	                #sFB_RightAngledTransfer421(iUDT_Configuration := #iUDT_Configuration."421".RightAngledTransfer,
	                                            iUDT_LowerConveyorConfiguration := #iUDT_Configuration."420".Conveyor,
	                                            iUDT_UpperConveyorConfiguration := #iUDT_Configuration."421".Conveyor,
	                                            iUDT_PECConfiguration := #iUDT_Configuration."420".PEC_EoS,
	                                            ii_DestinationA := 0,
	                                            ii_DestinationB := 0,
	                                            ii_DestinationC := 0,
	                                            ii_DestinationD := 1,
	                                            ix_HardwareOk := #iUDT_HardwareOk."420",
	                                            ix_400vOk := #ix_400vOk,
	                                            ix_24vOk := #ix_24vOk,
	                                            ix_SafetyOk := #ix_SafetyOk,
	                                            ix_AirPressureOk := #ix_AirPressureOk,
	                                            ix_SectionIsDown := #sFB_MCOConveyLinxAixController420.sUDT_AixInputsFullModule.AllSensorPortInputs.RightPin2,
	                                            ix_SectionIsUp := #sFB_MCOConveyLinxAixController420.sUDT_AixInputsFullModule.AllSensorPortInputs.RightSensor,
	                                            ix_ConveyorAAuto := FALSE,
	                                            ix_ConveyorBAuto := #iqUDT_WorkstationCommonStatus."430".AutoON,
	                                            ix_ConveyorCAuto := FALSE,
	                                            ix_ConveyorDAuto := #iqUDT_WorkstationCommonStatus."410".AutoON,
	                                            ix_PEC := #sFB_MCOConveyLinxAixController420.sUDT_AixInputsFullModule.AllSensorPortInputs.LeftSensor,
	                                            ix_ExternalReceiveRequestA := FALSE,
	                                            ix_ExternalReceiveRequestB := FALSE,
	                                            ix_ExternalReceiveRequestC := FALSE,
	                                            ix_ExternalReceiveRequestD := NOT #iqUDT_WorkstationStatus."410".PEC_EoS.PEC,
	                                            ix_PECInfeedA := false,
	                                            ix_PECInfeedD := #iqUDT_WorkstationStatus."410".PEC_EoS.PEC,
	                                            qUDT_HMIRATStatus => #iqUDT_WorkstationStatus."421".RightAngledTransfer,
	                                            qUDT_HMIConveyorStatus => #iqUDT_WorkstationStatus."420".Conveyor,
	                                            qUDT_HMIPECStatus => #iqUDT_WorkstationStatus."421".PEC_EoS,
	                                            qUDT_RATStatus => #iqUDT_WorkstationCommonStatus."421",
	                                            qUDT_ConveyorStatus => #iqUDT_WorkstationCommonStatus."420",
	                                            qx_PopupControl => #qx_PopupControl421,
	                                            qx_ExternalSendRequestA => #tx_dummy,
	                                            qx_ExternalSendRequestB => #tx_dummy,
	                                            qx_ExternalSendRequestC => #tx_dummy,
	                                            qx_ExternalSendRequestD => #tx_dummy,
	                                            iqUDT_EquipmentControl := #iqUDT_EquipmentControlFirstStation,
	                                            iqUDT_RATCommand := #iqUDT_WorkstationCommands."421".RightAngledTransfer,
	                                            iqUDT_ConveyorCommand := #iqUDT_WorkstationCommands."420".Conveyor,
	                                            iqUDT_RATStatistics := #iqUDT_WorkstationStatistics."421".RightAngledTransfer,
	                                            iqUDT_ConveyorStatistics := #iqUDT_WorkstationStatistics."420".Conveyor,
	                                            iqUDT_PECStatistics := #iqUDT_WorkstationStatistics."421".PEC_EoS,
	                                            iqUDT_HandShakeConveyorA := #tUDT_dummyHandshake,
	                                            iqUDT_HandShakeConveyorB := #sUDT_Handshake420,
	                                            iqUDT_HandShakeConveyorC := #tUDT_dummyHandshake,
	                                            iqUDT_HandShakeConveyorD := #sUDT_Handshake410,
	                                            iqUDT_LowerConveyorInterface := #sUDT_Interface420,
	                                            iqUDT_UpperConveyorInterface := #sUDT_Interface421,
	                                            iqUDT_RATPositioning := #iqUDT_RATPositioning420,
	                                            iqUDT_BladeStopEoSInterface := #tudt_Bladeinterfacedummy,
	                                            iqUDT_BladeStopBoSInterface := #tudt_Bladeinterfacedummy);

	            END_REGION

	            REGION MCO

	                #sFB_MCOConveyLinxAixController421(iUDT_AixConfig := #iUDT_Configuration."421".MCO_M01,
	                                                   iv_AixInputsModule := #iv_MotorInput420,
	                                                   ii_PositionSetpoint := #iqUDT_RATPositioning420.Upper.EndPosition,
	                                                   ix_24vOk := #ix_24vOk,
	                                                   ix_SimulationModeActive := "DB_Memory".Simulation,
	                                                   ii_MotorPositionId := 2,
	                                                   ix_StartPositioning := #iqUDT_RATPositioning420.Upper.Start,
	                                                   ix_ResetPosition := #iqUDT_RATPositioning420.Upper.ResetPosition,
	                                                   qUDT_HMIStatus => #iqUDT_WorkstationStatus."421".MCO_M01,
	                                                   qx_Positioned => #iqUDT_RATPositioning420.Upper.Done,
	                                                   iqv_AixOutputsModule := #iqv_MotorOutput420,
	                                                   iqUDT_ConveyorInterface := #sUDT_Interface421,
	                                                   iqUDT_MCOStatistics := #iqUDT_WorkstationStatistics."421".MCO_M01);
	            END_REGION

	        END_REGION

	        REGION 430
	            REGION ZPA First conveyor

	                #sFB_ZpaFirstConveyor430(iUDT_AixInputsModule := #iUDT_InputsModule430,
	                                         iUDT_AixZpaConfig := #iUDT_Configuration."430".Conveyor,
	                                       ix_24vOk := NOT #ix_24vOk,
	                                       ix_HardwareOk := #iUDT_HardwareOk."430",
	                                       ix_SimulationModeActive := "DB_Memory".Simulation,
	                                       qUDT_AixOutputsModule => #qUDT_OutputsModule430,
	                                       iqUDT_ZPAinterface := #sUDT_ZPAinterface430,
	                                       iqUDT_PecStatus := #iqUDT_WorkstationStatus."430".PEC_EoS,
	                                       iqUDT_ZpaControllerStatus := #iqUDT_WorkstationStatus."430".MCO_ZPA,
	                                       iqUDT_HandShakeUp := #sUDT_Handshake430);
	            END_REGION

	            REGION ZPA Zone status

	                #sFB_ZpaStatus430(ii_ModuleID := 1,
	                                        iqUDT_PecStatus := #iqUDT_WorkstationStatus."430".PEC_EoS,
	                                        iqUDT_ZpaControllerStatus := #iqUDT_WorkstationStatus."430".MCO_ZPA,
	                                        iqUDT_ZPAInterface := #sUDT_ZPAinterface430,
	                                        qUDT_ConveyorStatus => #iqUDT_WorkstationStatus."430".Conveyor);

	            END_REGION
	        END_REGION

	        REGION 440
	            REGION ZPA Zone status

	                #sFB_ZpaStatus440(ii_ModuleID := 1,
	                                        iqUDT_PecStatus := #iqUDT_WorkstationStatus."440".PEC_EoS,
	                                        iqUDT_ZpaControllerStatus := #iqUDT_WorkstationStatus."440".MCO_ZPA,
	                                        iqUDT_ZPAInterface := #sUDT_ZPAinterface430,
	                                        qUDT_ConveyorStatus => #iqUDT_WorkstationStatus."440".Conveyor);

	            END_REGION
	        END_REGION

	        REGION 450
	            REGION ZPA Zone status

	                #sFB_ZpaStatus450(ii_ModuleID := 2,
	                                        iqUDT_PecStatus := #iqUDT_WorkstationStatus."450".PEC_EoS,
	                                        iqUDT_ZpaControllerStatus := #iqUDT_WorkstationStatus."450".MCO_ZPA,
	                                        iqUDT_ZPAInterface := #sUDT_ZPAinterface430,
	                                        qUDT_ConveyorStatus => #iqUDT_WorkstationStatus."450".Conveyor);

	            END_REGION
	        END_REGION

	        REGION 260
	            REGION ZPA Zone status

	                #sFB_ZpaStatus460(ii_ModuleID := 2,
	                                        iqUDT_PecStatus := #iqUDT_WorkstationStatus."260".PEC_EoS,
	                                        iqUDT_ZpaControllerStatus := #iqUDT_WorkstationStatus."260".MCO_ZPA,
	                                        iqUDT_ZPAInterface := #sUDT_ZPAinterface230,
	                                        qUDT_ConveyorStatus => #iqUDT_WorkstationStatus."260".Conveyor);

	            END_REGION
	        END_REGION

	        REGION 470
	            REGION ZPA Zone status

	                #sFB_ZpaStatus470(ii_ModuleID := 3,
	                                        iqUDT_PecStatus := #iqUDT_WorkstationStatus."470".PEC_EoS,
	                                        iqUDT_ZpaControllerStatus := #iqUDT_WorkstationStatus."470".MCO_ZPA,
	                                        iqUDT_ZPAInterface := #sUDT_ZPAinterface430,
	                                        qUDT_ConveyorStatus => #iqUDT_WorkstationStatus."470".Conveyor);

	            END_REGION
	        END_REGION

	        REGION 480
	            REGION ZPA Last conveyor

	                #sFB_ZpaLastConveyor480(iUDT_AixInputsModule := #iUDT_InputsModule470,
	                                        iUDT_AixZpaConfig := #iUDT_Configuration."480".Conveyor,
	                                      ix_SafetyOk := #ix_SafetyOk,
	                                      ix_24vOk := #ix_24vOk,
	                                      ix_HardwareOk := #iUDT_HardwareOk."480",
	                                      ix_SimulationModeActive := "DB_Memory".Simulation,
	                                      qUDT_AixOutputsModule => #qUDT_OutputsModule470,
	                                      qUDT_CommonStatus => #iqUDT_WorkstationCommonStatus."480",
	                                      iqUDT_EquipmentControl := #iqUDT_EquipmentControlSecondStation,
	                                      iqUDT_ZPACommand := #iqUDT_WorkstationCommands."480".SegmentZPA,
	                                      iqUDT_ZPAinterface := #sUDT_ZPAinterface430,
	                                      iqUDT_PecStatus := #iqUDT_WorkstationStatus."480".PEC_EoS,
	                                      iqUDT_ZpaControllerStatus := #iqUDT_WorkstationStatus."480".MCO_ZPA,
	                                      iqUDT_Handshake := #sUDT_Handshake480);
	            END_REGION

	            REGION ZPA Zone status

	                #sFB_ZpaStatus480(ii_ModuleID := 3,
	                                        iqUDT_PecStatus := #iqUDT_WorkstationStatus."280".PEC_EoS,
	                                        iqUDT_ZpaControllerStatus := #iqUDT_WorkstationStatus."280".MCO_ZPA,
	                                        iqUDT_ZPAInterface := #sUDT_ZPAinterface230,
	                                        qUDT_ConveyorStatus => #iqUDT_WorkstationStatus."280".Conveyor);

	            END_REGION

	            REGION Barcode Scanner
	                #sFB_Scanner_481(iUDT_ScannerInput := #iUDT_ScannerInput501,
	                                 iUDT_ScannerConfiguration := #iUDT_Configuration."481",
	                                 iUDT_ConveyorInterface := #sUDT_Interface480,
	                                 ix_24vOk := TRUE,
	                                 ix_HardwareOk := TRUE,
	                                 ix_SimulationModeActive := FALSE,
	                                 ix_CloseWindow := #iqUDT_WorkstationStatus."480".PEC_EoS.PEC,
	                                 ix_Trigger := NOT #iqUDT_WorkstationStatus."480".PEC_EoS.PEC,
	                                 qUDT_ScannerOutput => #qUDT_ScannerOutput501,
	                                 qUDT_HMIStatus => #iqUDT_WorkstationStatus."481",
	                                 qUDT_CommonStatus => #iqUDT_WorkstationCommonStatus."481",
	                                 qs_Barcode => #ts_Barcode481,
	                                 iqUDT_Statistics := #iqUDT_WorkstationStatistics."481",
	                                 iqUDT_EquipmentControl := #iqUDT_EquipmentControlSecondStation);
	            END_REGION
	        END_REGION

	        REGION 490

	            REGION Displacement
	                #sFB_Displacement490(#sUDT_Interface490);
	            END_REGION

	            REGION MCO

	                #sFB_MCOConveyLinxAixController490(iUDT_AixConfig := #iUDT_Configuration."490".MCO_M01,
	                                                   iv_AixInputsModule := #iv_MotorInput490,
	                                                   ii_PositionSetpoint := #iqUDT_RATPositioning490.Lower.EndPosition,
	                                                   ix_24vOk := #ix_24vOk,
	                                                   ix_SimulationModeActive := "DB_Memory".Simulation,
	                                                   ii_MotorPositionId := 1,
	                                                   ix_StartPositioning := #iqUDT_RATPositioning490.Lower.Start,
	                                                   ix_ResetPosition := #iqUDT_RATPositioning490.Lower.ResetPosition,
	                                                   qUDT_HMIStatus => #iqUDT_WorkstationStatus."490".MCO_M01,
	                                                   qx_Positioned => #iqUDT_RATPositioning490.Lower.Done,
	                                                   iqv_AixOutputsModule := #iqv_MotorOutput490,
	                                                   iqUDT_ConveyorInterface := #sUDT_Interface490,
	                                                   iqUDT_MCOStatistics := #iqUDT_WorkstationStatistics."490".MCO_M01);
	            END_REGION
	        END_REGION


	        REGION 491

	            REGION Displacement
	                #sFB_Displacement491(#sUDT_Interface491);
	            END_REGION

	            REGION RAT

	                #sFB_RightAngledTransfer491(iUDT_Configuration := #iUDT_Configuration."491".RightAngledTransfer,
	                                            iUDT_LowerConveyorConfiguration := #iUDT_Configuration."490".Conveyor,
	                                            iUDT_UpperConveyorConfiguration := #iUDT_Configuration."491".Conveyor,
	                                            iUDT_PECConfiguration := #iUDT_Configuration."490".PEC_EoS,
	                                            ii_DestinationA := #si_DestinationA491,
	                                            ii_DestinationB := 0,
	                                            ii_DestinationC := 0,
	                                            ii_DestinationD := 0,
	                                            ix_HardwareOk := #iUDT_HardwareOk."490",
	                                            ix_400vOk := #ix_400vOk,
	                                            ix_24vOk := #ix_24vOk,
	                                            ix_SafetyOk := #ix_SafetyOk,
	                                            ix_AirPressureOk := #ix_AirPressureOk,
	                                            ix_SectionIsDown := #sFB_MCOConveyLinxAixController490.sUDT_AixInputsFullModule.AllSensorPortInputs.RightPin2,
	                                            ix_SectionIsUp := #sFB_MCOConveyLinxAixController490.sUDT_AixInputsFullModule.AllSensorPortInputs.RightSensor,
	                                            ix_ConveyorAAuto := #iqUDT_WorkstationCommonStatus."480".AutoON,
	                                            ix_ConveyorBAuto := FALSE,
	                                            ix_ConveyorCAuto := FALSE,
	                                            ix_ConveyorDAuto := #iqUDT_WorkstationCommonStatus."500".AutoON,
	                                            ix_PEC := #sFB_MCOConveyLinxAixController490.sUDT_AixInputsFullModule.AllSensorPortInputs.LeftSensor,
	                                            ix_ExternalReceiveRequestA := NOT #iqUDT_WorkstationStatus."480".PEC_EoS.PEC,
	                                            ix_ExternalReceiveRequestB := FALSE,
	                                            ix_ExternalReceiveRequestC := FALSE,
	                                            ix_ExternalReceiveRequestD := FALSE,
	                                            ix_PECInfeedA := #iqUDT_WorkstationStatus."480".PEC_EoS.PEC,
	                                            qUDT_HMIRATStatus => #iqUDT_WorkstationStatus."491".RightAngledTransfer,
	                                            qUDT_HMIConveyorStatus => #iqUDT_WorkstationStatus."490".Conveyor,
	                                            qUDT_HMIPECStatus => #iqUDT_WorkstationStatus."491".PEC_EoS,
	                                            qUDT_RATStatus => #iqUDT_WorkstationCommonStatus."491",
	                                            qUDT_ConveyorStatus => #iqUDT_WorkstationCommonStatus."490",
	                                            qx_PopupControl => #qx_PopupControl491,
	                                            qx_ExternalSendRequestA => #tx_dummy,
	                                            qx_ExternalSendRequestB => #tx_dummy,
	                                            qx_ExternalSendRequestC => #tx_dummy,
	                                            qx_ExternalSendRequestD => #tx_dummy,
	                                            iqUDT_EquipmentControl := #iqUDT_EquipmentControlFirstStation,
	                                            iqUDT_RATCommand := #iqUDT_WorkstationCommands."491".RAT,
	                                            iqUDT_ConveyorCommand := #iqUDT_WorkstationCommands."490".Conveyor,
	                                            iqUDT_RATStatistics := #iqUDT_WorkstationStatistics."491".RightAngledTransfer,
	                                            iqUDT_ConveyorStatistics := #iqUDT_WorkstationStatistics."490".Conveyor,
	                                            iqUDT_PECStatistics := #iqUDT_WorkstationStatistics."491".PEC_EoS,
	                                            iqUDT_HandShakeConveyorA := #sUDT_Handshake480,
	                                            iqUDT_HandShakeConveyorB := #tUDT_dummyHandshake,
	                                            iqUDT_HandShakeConveyorC := #tUDT_dummyHandshake,
	                                            iqUDT_HandShakeConveyorD := #sUDT_Handshake491,
	                                            iqUDT_LowerConveyorInterface := #sUDT_Interface490,
	                                            iqUDT_UpperConveyorInterface := #sUDT_Interface491,
	                                            iqUDT_RATPositioning := #iqUDT_RATPositioning490,
	                                            iqUDT_BladeStopEoSInterface := #tudt_Bladeinterfacedummy,
	                                            iqUDT_BladeStopBoSInterface := #tudt_Bladeinterfacedummy);



	            END_REGION

	            REGION MCO

	                #sFB_MCOConveyLinxAixController491(iUDT_AixConfig := #iUDT_Configuration."491".MCO_M01,
	                                                   iv_AixInputsModule := #iv_MotorInput490,
	                                                   ix_24vOk := #ix_24vOk,
	                                                   ix_SimulationModeActive := "DB_Memory".Simulation,
	                                                   ii_MotorPositionId := 2,
	                                                   qUDT_HMIStatus => #iqUDT_WorkstationStatus."491".MCO_M01,
	                                                   iqv_AixOutputsModule := #iqv_MotorOutput490,
	                                                   iqUDT_ConveyorInterface := #sUDT_Interface491,
	                                                   iqUDT_MCOStatistics := #iqUDT_WorkstationStatistics."491".MCO_M01);
	            END_REGION

	        END_REGION

	        REGION 500

	            REGION Displacement
	                #sFB_Displacement500(#sUDT_Interface500);
	            END_REGION

	            REGION EoS

	                #sFB_PEC500(ix_PEC := #sFB_MCOConveyLinxAixController500.sUDT_AixInputsFullModule.AllSensorPortInputs.LeftSensor,
	                            iUDT_PECConfiguration := #iUDT_Configuration."500".PEC_EoS,
	                            qUDT_HMIStatus => #iqUDT_WorkstationStatus."500".PEC_EoS,
	                            iqUDT_ConveyorInterface := #sUDT_Interface500,
	                            iqUDT_PECStatistics := #iqUDT_WorkstationStatistics."500".PEC_EoS);

	            END_REGION
	            REGION Conveyor

	                // IF #sUDT_Handshake500.TIP OR (#sFB_RightAngledTransfer491.sx_UpperTransportOut AND NOT #iqUDT_WorkstationStatus."491".PEC.PEC)
	                // THEN
	                //     #ti_externalSpeed_500 := #iUDT_Configuration."500".Conveyor.SpeedSetpointNominal;
	                // ELSE
	                //     #ti_externalSpeed_500 := #iUDT_Configuration."500".Conveyor.SpeedSetpointNominal / 2;
	                // END_IF;

	                #sUDT_Handshake500.RTR := #sUDT_Handshake500.RTR OR #iqUDT_WorkstationStatus."500".PEC_EoS.PEC;

	                #sFB_Conveyor500(iUDT_ConveyorConfiguration := #iUDT_Configuration."500".Conveyor,
	                                 idi_PECEoSDistance := #iUDT_Configuration."500".PEC_EoS.Distance,
	                                 idi_PECBoSDistance := 0,
	                                 ii_ExternalSpeed := #ti_externalSpeed_500,
	                                 ix_SafetyOk := #ix_SafetyOk,
	                                 ix_24vOk := #ix_24vOk,
	                                 ix_400vOk := #ix_400vOk,
	                                 ix_HardwareOk := #iUDT_HardwareOk."500",
	                                 ix_PECEoS := #iqUDT_WorkstationStatus."500".PEC_EoS.PEC,
	                                 ix_PECBoS := TRUE,
	                                 ix_ReverseDirection := FALSE,
	                                 ix_ExternalRequestDieBack := FALSE,
	                                 ix_ExternalRequestHold := #iqUDT_WorkstationStatus."611".PEC_EoS.Jam,
	                                 ix_ResetEnergySave := FALSE,
	                                 qUDT_HMIStatus => #iqUDT_WorkstationStatus."500".Conveyor,
	                                 qUDT_Status => #iqUDT_WorkstationCommonStatus."500",
	                                 iqUDT_EquipmentControl := #iqUDT_EquipmentControlFirstStation,
	                                 iqUDT_ConveyorCommand := #iqUDT_WorkstationCommands."500".Conveyor,
	                                 iqUDT_ConveyorInterface := #sUDT_Interface500,
	                                 iqUDT_HandShakeUp := #sUDT_Handshake491,
	                                 iqUDT_HandShake := #sUDT_Handshake500,
	                                 iqUDT_Statistics := #iqUDT_WorkstationStatistics."500".Conveyor);

	            END_REGION
	            REGION MCO

	                #sFB_MCOConveyLinxAixController500(iUDT_AixConfig := #iUDT_Configuration."500".MCO_M01,
	                                                   iv_AixInputsModule := #iv_MotorInput500,
	                                                   ix_24vOk := #ix_24vOk,
	                                                   ix_SimulationModeActive := "DB_Memory".Simulation,
	                                                   ii_MotorPositionId := 1,
	                                                   qUDT_HMIStatus => #iqUDT_WorkstationStatus."500".MCO_M01,
	                                                   iqv_AixOutputsModule := #iqv_MotorOutput500,
	                                                   iqUDT_ConveyorInterface := #sUDT_Interface500,
	                                                   iqUDT_MCOStatistics := #iqUDT_WorkstationStatistics."500".MCO_M01);
	            END_REGION
	        END_REGION
	    END_IF;
	END_REGION

	REGION 6 - Station Outfeed
	    REGION 610

	        REGION Displacement
	            #sFB_Displacement610(#sUDT_Interface610);
	        END_REGION

	        REGION MCO

	            #sFB_MCOConveyLinxAixController610(iUDT_AixConfig := #iUDT_Configuration."610".MCO_M01,
	                                               iv_AixInputsModule := #iv_MotorInput610,
	                                               ix_24vOk := #ix_24vOk,
	                                               ix_SimulationModeActive := "DB_Memory".Simulation,
	                                               ii_MotorPositionId := 1,
	                                               qUDT_HMIStatus => #iqUDT_WorkstationStatus."610".MCO_M01,
	                                               iqv_AixOutputsModule := #iqv_MotorOutput610,
	                                               iqUDT_ConveyorInterface := #sUDT_Interface610,
	                                               iqUDT_MCOStatistics := #iqUDT_WorkstationStatistics."610".MCO_M01);
	        END_REGION
	    END_REGION

	    REGION 611



	        REGION Displacement
	            #sFB_Displacement611(#sUDT_Interface611);
	        END_REGION

	        REGION RAT

	            #sFB_RightAngledTransfer611(iUDT_Configuration := #iUDT_Configuration."611".RightAngledTransfer,
	                                        iUDT_LowerConveyorConfiguration := #iUDT_Configuration."610".Conveyor,
	                                        iUDT_UpperConveyorConfiguration := #iUDT_Configuration."611".Conveyor,
	                                        iUDT_PECConfiguration := #iUDT_Configuration."610".PEC_EoS,
	                                        ii_DestinationA := 0,
	                                        ii_DestinationB := 0,
	                                        ii_DestinationC := 1,
	                                        ii_DestinationD := 1,
	                                        ix_HardwareOk := #iUDT_HardwareOk."610",
	                                        ix_400vOk := #ix_400vOk,
	                                        ix_24vOk := #ix_24vOk,
	                                        ix_SafetyOk := #ix_SafetyOk,
	                                        ix_AirPressureOk := #ix_AirPressureOk,
	                                        ix_SectionIsDown := #sFB_MCOConveyLinxAixController610.sUDT_AixInputsFullModule.AllSensorPortInputs.RightPin2,
	                                        ix_SectionIsUp := #sFB_MCOConveyLinxAixController610.sUDT_AixInputsFullModule.AllSensorPortInputs.RightSensor,
	                                        ix_ConveyorAAuto := TRUE,
	                                        ix_ConveyorBAuto := #iqUDT_WorkstationCommonStatus."620".AutoON,
	                                        ix_ConveyorCAuto := #iqUDT_WorkstationCommonStatus."500".AutoON,
	                                        ix_ConveyorDAuto := #iqUDT_WorkstationCommonStatus."300".AutoON,
	                                        ix_PEC := #sFB_MCOConveyLinxAixController610.sUDT_AixInputsFullModule.AllSensorPortInputs.LeftSensor,
	                                        ix_ExternalReceiveRequestA := FALSE,
	                                        ix_ExternalReceiveRequestB := FALSE,
	                                        ix_ExternalReceiveRequestC := NOT #iqUDT_WorkstationStatus."500".PEC_EoS.PEC,
	                                        ix_ExternalReceiveRequestD := NOT #iqUDT_WorkstationStatus."300".PEC_EoS.PEC,
	                                        ix_PECInfeedC := #iqUDT_WorkstationStatus."500".PEC_EoS.PEC,
	                                        ix_PECInfeedD := #iqUDT_WorkstationStatus."300".PEC_EoS.PEC,
	                                        qUDT_HMIRATStatus => #iqUDT_WorkstationStatus."611".RightAngledTransfer,
	                                        qUDT_HMIConveyorStatus => #iqUDT_WorkstationStatus."610".Conveyor,
	                                        qUDT_HMIPECStatus => #iqUDT_WorkstationStatus."611".PEC_EoS,
	                                        qUDT_RATStatus => #iqUDT_WorkstationCommonStatus."611",
	                                        qUDT_ConveyorStatus => #iqUDT_WorkstationCommonStatus."610",
	                                        qx_PopupControl => #qx_PopupControl611,
	                                        qx_ExternalSendRequestA => #tx_dummy,
	                                        qx_ExternalSendRequestB => #tx_dummy,
	                                        qx_ExternalSendRequestC => #tx_dummy,
	                                        qx_ExternalSendRequestD => #tx_dummy,
	                                        iqUDT_EquipmentControl := #iqUDT_EquipmentControlInfeed,
	                                        iqUDT_RATCommand := #iqUDT_WorkstationCommands."611".RightAngledTransfer,
	                                        iqUDT_ConveyorCommand := #iqUDT_WorkstationCommands."610".Conveyor,
	                                        iqUDT_RATStatistics := #iqUDT_WorkstationStatistics."611".RightAngledTransfer,
	                                        iqUDT_ConveyorStatistics := #iqUDT_WorkstationStatistics."610".Conveyor,
	                                        iqUDT_PECStatistics := #iqUDT_WorkstationStatistics."611".PEC_EoS,
	                                        iqUDT_HandShakeConveyorA := #tUDT_dummyHandshake,
	                                        iqUDT_HandShakeConveyorB := #sUDT_Handshake610,
	                                        iqUDT_HandShakeConveyorC := #sUDT_Handshake500,
	                                        iqUDT_HandShakeConveyorD := #sUDT_Handshake300,
	                                        iqUDT_LowerConveyorInterface := #sUDT_Interface610,
	                                        iqUDT_UpperConveyorInterface := #sUDT_Interface611,
	                                        iqUDT_RATPositioning := #iqUDT_RATPositioning610,
	                                        iqUDT_BladeStopEoSInterface := #tudt_Bladeinterfacedummy,
	                                        iqUDT_BladeStopBoSInterface := #tudt_Bladeinterfacedummy);

	        END_REGION

	        REGION MCO

	            #sFB_MCOConveyLinxAixController611(iUDT_AixConfig := #iUDT_Configuration."611".MCO_M01,
	                                               iv_AixInputsModule := #iv_MotorInput610,
	                                               ii_PositionSetpoint := #iqUDT_RATPositioning610.Upper.EndPosition,
	                                               ix_24vOk := #ix_24vOk,
	                                               ix_SimulationModeActive := "DB_Memory".Simulation,
	                                               ii_MotorPositionId := 2,
	                                               ix_StartPositioning := #iqUDT_RATPositioning610.Upper.Start,
	                                               ix_ResetPosition := #iqUDT_RATPositioning610.Upper.ResetPosition,
	                                               qUDT_HMIStatus => #iqUDT_WorkstationStatus."611".MCO_M01,
	                                               qx_Positioned => #iqUDT_RATPositioning610.Upper.Done,
	                                               iqv_AixOutputsModule := #iqv_MotorOutput610,
	                                               iqUDT_ConveyorInterface := #sUDT_Interface611,
	                                               iqUDT_MCOStatistics := #iqUDT_WorkstationStatistics."611".MCO_M01);
	        END_REGION

	    END_REGION

	    REGION 620

	        REGION Displacement
	            #sFB_Displacement620(#sUDT_Interface620);
	        END_REGION
	        REGION EoS

	            #sFB_PEC620(ix_PEC := #sFB_MCOConveyLinxAixController620.sUDT_AixInputsFullModule.AllSensorPortInputs.LeftSensor,
	                        iUDT_PECConfiguration := #iUDT_Configuration."620".PEC_EoS,
	                        qUDT_HMIStatus => #iqUDT_WorkstationStatus."620".PEC_EoS,
	                        iqUDT_ConveyorInterface := #sUDT_Interface620,
	                        iqUDT_PECStatistics := #iqUDT_WorkstationStatistics."620".PEC_EoS);

	        END_REGION

	        REGION Conveyor

	            #sFB_Conveyor620(iUDT_ConveyorConfiguration := #iUDT_Configuration."620".Conveyor,
	                             idi_PECEoSDistance := 0,
	                             idi_PECBoSDistance := 0,
	                             ii_ExternalSpeed := 0,
	                             ix_SafetyOk := #ix_SafetyOk,
	                             ix_24vOk := #ix_24vOk,
	                             ix_400vOk := #ix_400vOk,
	                             ix_HardwareOk := #iUDT_HardwareOk."620",
	                             ix_PECEoS := #iqUDT_WorkstationStatus."620".PEC_EoS.PEC,
	                             ix_PECBoS := TRUE,
	                             ix_ReverseDirection := FALSE,
	                             ix_ExternalRequestDieBack := FALSE,
	                             ix_ExternalRequestHold := FALSE,
	                             ix_ResetEnergySave := FALSE,
	                             qUDT_HMIStatus => #iqUDT_WorkstationStatus."620".Conveyor,
	                             qUDT_Status => #iqUDT_WorkstationCommonStatus."620",
	                             iqUDT_EquipmentControl := #iqUDT_EquipmentControlFirstStation,
	                             iqUDT_ConveyorCommand := #iqUDT_WorkstationCommands."620".Conveyor,
	                             iqUDT_ConveyorInterface := #sUDT_Interface620,
	                             iqUDT_HandShakeUp := #sUDT_Handshake610,
	                             iqUDT_HandShake := #sUDT_Handshake620,
	                             iqUDT_Statistics := #iqUDT_WorkstationStatistics."620".Conveyor);

	        END_REGION

	        REGION MCO

	            #sFB_MCOConveyLinxAixController620(iUDT_AixConfig := #iUDT_Configuration."620".MCO_M01,
	                                               iv_AixInputsModule := #iv_MotorInput620,
	                                               ix_24vOk := #ix_24vOk,
	                                               ix_SimulationModeActive := "DB_Memory".Simulation,
	                                               ii_MotorPositionId := 1,
	                                               qUDT_HMIStatus => #iqUDT_WorkstationStatus."620".MCO_M01,
	                                               iqv_AixOutputsModule := #iqv_MotorOutput620,
	                                               iqUDT_ConveyorInterface := #sUDT_Interface620,
	                                               iqUDT_MCOStatistics := #iqUDT_WorkstationStatistics."620".MCO_M01);
	        END_REGION

	    END_REGION

	    REGION 630

	        REGION Displacement
	            #sFB_Displacement630(#sUDT_Interface630);
	        END_REGION

	        REGION EoS

	            #sFB_PEC630(ix_PEC := #sFB_MCOConveyLinxAixController630.sUDT_AixInputsFullModule.AllSensorPortInputs.LeftSensor,
	                        iUDT_PECConfiguration := #iUDT_Configuration."630".PEC_EoS,
	                        qUDT_HMIStatus => #iqUDT_WorkstationStatus."630".PEC_EoS,
	                        iqUDT_ConveyorInterface := #sUDT_Interface630,
	                        iqUDT_PECStatistics := #iqUDT_WorkstationStatistics."630".PEC_EoS);

	        END_REGION

	        REGION Conveyor

	            #sFB_Conveyor630(iUDT_ConveyorConfiguration := #iUDT_Configuration."630".Conveyor,
	                             idi_PECEoSDistance := 0,
	                             idi_PECBoSDistance := 0,
	                             ii_ExternalSpeed := 0,
	                             ix_SafetyOk := #ix_SafetyOk,
	                             ix_24vOk := #ix_24vOk,
	                             ix_400vOk := #ix_400vOk,
	                             ix_HardwareOk := #iUDT_HardwareOk."630",
	                             ix_PECEoS := #iqUDT_WorkstationStatus."630".PEC_EoS.PEC,
	                             ix_PECBoS := TRUE,
	                             ix_ReverseDirection := FALSE,
	                             ix_ExternalRequestDieBack := FALSE,
	                             ix_ExternalRequestHold := FALSE,
	                             ix_ResetEnergySave := FALSE,
	                             qUDT_HMIStatus => #iqUDT_WorkstationStatus."630".Conveyor,
	                             qUDT_Status => #iqUDT_WorkstationCommonStatus."630",
	                             iqUDT_EquipmentControl := #iqUDT_EquipmentControlFirstStation,
	                             iqUDT_ConveyorCommand := #iqUDT_WorkstationCommands."630".Conveyor,
	                             iqUDT_ConveyorInterface := #sUDT_Interface630,
	                             iqUDT_HandShakeUp := #sUDT_Handshake620,
	                             iqUDT_HandShake := #sUDT_Handshake630,
	                             iqUDT_Statistics := #iqUDT_WorkstationStatistics."630".Conveyor);

	        END_REGION

	        REGION MCO

	            #sFB_MCOConveyLinxAixController630(iUDT_AixConfig := #iUDT_Configuration."630".MCO_M01,
	                                               iv_AixInputsModule := #iv_MotorInput630,
	                                               ix_24vOk := #ix_24vOk,
	                                               ix_SimulationModeActive := "DB_Memory".Simulation,
	                                               ii_MotorPositionId := 1,
	                                               qUDT_HMIStatus => #iqUDT_WorkstationStatus."630".MCO_M01,
	                                               iqv_AixOutputsModule := #iqv_MotorOutput630,
	                                               iqUDT_ConveyorInterface := #sUDT_Interface630,
	                                               iqUDT_MCOStatistics := #iqUDT_WorkstationStatistics."630".MCO_M01);
	        END_REGION
	    END_REGION

	    REGION 640

	        REGION Displacement
	            #sFB_Displacement640(#sUDT_Interface640);
	        END_REGION

	        REGION EoS

	            #sFB_PEC640(ix_PEC := #sFB_MCOConveyLinxAixController640.sUDT_AixInputsFullModule.AllSensorPortInputs.LeftSensor,
	                        iUDT_PECConfiguration := #iUDT_Configuration."640".PEC_EoS,
	                        qUDT_HMIStatus => #iqUDT_WorkstationStatus."640".PEC_EoS,
	                        iqUDT_ConveyorInterface := #sUDT_Interface640,
	                        iqUDT_PECStatistics := #iqUDT_WorkstationStatistics."640".PEC_EoS);

	        END_REGION
	        REGION Conveyor

	            #sFB_Conveyor640(iUDT_ConveyorConfiguration := #iUDT_Configuration."640".Conveyor,
	                             idi_PECEoSDistance := #iUDT_Configuration."640".PEC_EoS.Distance,
	                             idi_PECBoSDistance := 0,
	                             ii_ExternalSpeed := 0,
	                             ix_SafetyOk := #ix_SafetyOk,
	                             ix_24vOk := #ix_24vOk,
	                             ix_400vOk := #ix_400vOk,
	                             ix_HardwareOk := #iUDT_HardwareOk."640",
	                             ix_PECEoS := #iqUDT_WorkstationStatus."640".PEC_EoS.PEC,
	                             ix_PECBoS := TRUE,
	                             ix_ReverseDirection := FALSE,
	                             ix_ExternalRequestDieBack := FALSE,
	                             ix_ExternalRequestHold := FALSE,
	                             ix_ResetEnergySave := FALSE,
	                             qUDT_HMIStatus => #iqUDT_WorkstationStatus."640".Conveyor,
	                             qUDT_Status => #iqUDT_WorkstationCommonStatus."640",
	                             iqUDT_EquipmentControl := #iqUDT_EquipmentControlFirstStation,
	                             iqUDT_ConveyorCommand := #iqUDT_WorkstationCommands."640".Conveyor,
	                             iqUDT_ConveyorInterface := #sUDT_Interface640,
	                             iqUDT_HandShakeUp := #sUDT_Handshake630,
	                             iqUDT_HandShake := #iqUDT_HandshakeDownstream640,
	                             iqUDT_Statistics := #iqUDT_WorkstationStatistics."640".Conveyor);

	        END_REGION

	        REGION MCO

	            #sFB_MCOConveyLinxAixController640(iUDT_AixConfig := #iUDT_Configuration."640".MCO_M01,
	                                               iv_AixInputsModule := #iv_MotorInput640,
	                                               ix_24vOk := #ix_24vOk,
	                                               ix_SimulationModeActive := "DB_Memory".Simulation,
	                                               ii_MotorPositionId := 1,
	                                               qUDT_HMIStatus => #iqUDT_WorkstationStatus."640".MCO_M01,
	                                               iqv_AixOutputsModule := #iqv_MotorOutput640,
	                                               iqUDT_ConveyorInterface := #sUDT_Interface640,
	                                               iqUDT_MCOStatistics := #iqUDT_WorkstationStatistics."640".MCO_M01);
	        END_REGION
	    END_REGION
	END_REGION


END_FUNCTION_BLOCK

